FUNCTION_BLOCK "G274M_Code"
TITLE =G274M EXHAUST AIR LOUVER KILN 1
//COPYRIGHT:    (C) 2009  BUHLER AG, CH-9240 UZWIL, SWITZERLAND
//
//PRODUCT:      WinCoS_BIW01_09
//
//TITLE:        EXHAUST AIR LOUVER KILN 1
//                Machine group control
//                Maschinengruppensteuerung
//
//--------------------------------------------------------------------------------
//
//IDENT:        AUTHOR:             DEPT:                              DATE:
//
//P01_FB374.1.0 K.Renz              CSB41                              30.Sep.2009
//             1st Release
//
//--------------------------------------------------------------------------------
//
//PURPOSE:
//
//MANUAL :
//
//RESTRICTIONS:
//
//--------------------------------------------------------------------------------
AUTHOR : KR
FAMILY : USW
VERSION : 9.9


VAR
  Gr : "GCS7_GrpCtrlSub";	//Standard interface to group
  InOutValue1 : DINT ;	//Data for user
  InOutValue2 : DINT ;	//Data for user
  OutWayConflict : BOOL ;	//Data for user
  OutSelectionOk : BOOL ;	//Data for user
  CmdNewValue : BOOL ;	//Data for user
  CmdNewJob : BOOL ;	//Data for user
  OutCodeOK : BOOL ;	//Data for user
  InEndOfJob : BOOL ;	//Data for user
  staWayOk : BOOL ;	//Data for user
  EdgeStartRelease : BOOL ;	//Data for user
  USW8 : BOOL ;	//Data for user
  USW9 : BOOL ;	//Data for user
  USW10 : BOOL ;	//Data for user
  USW11 : BOOL ;	//Data for user
  USW12 : BOOL ;	//Data for user
  USW13 : BOOL ;	//Data for user
  USW14 : BOOL ;	//Data for user
  USW15 : BOOL ;	//Data for user
END_VAR
VAR_TEMP
  tmpEnable : BOOL ;
  tmpFlag : BOOL ;
  tmpCmdNext : BOOL ;
  tmpLocal : BOOL ;
  tmpAspOk : BOOL ;
  tmpHWStop : BOOL ;
  tmpInstanzDBNo : INT ;
END_VAR
BEGIN
NETWORK
TITLE =



NETWORK
TITLE =Read command from group control
//Parameter
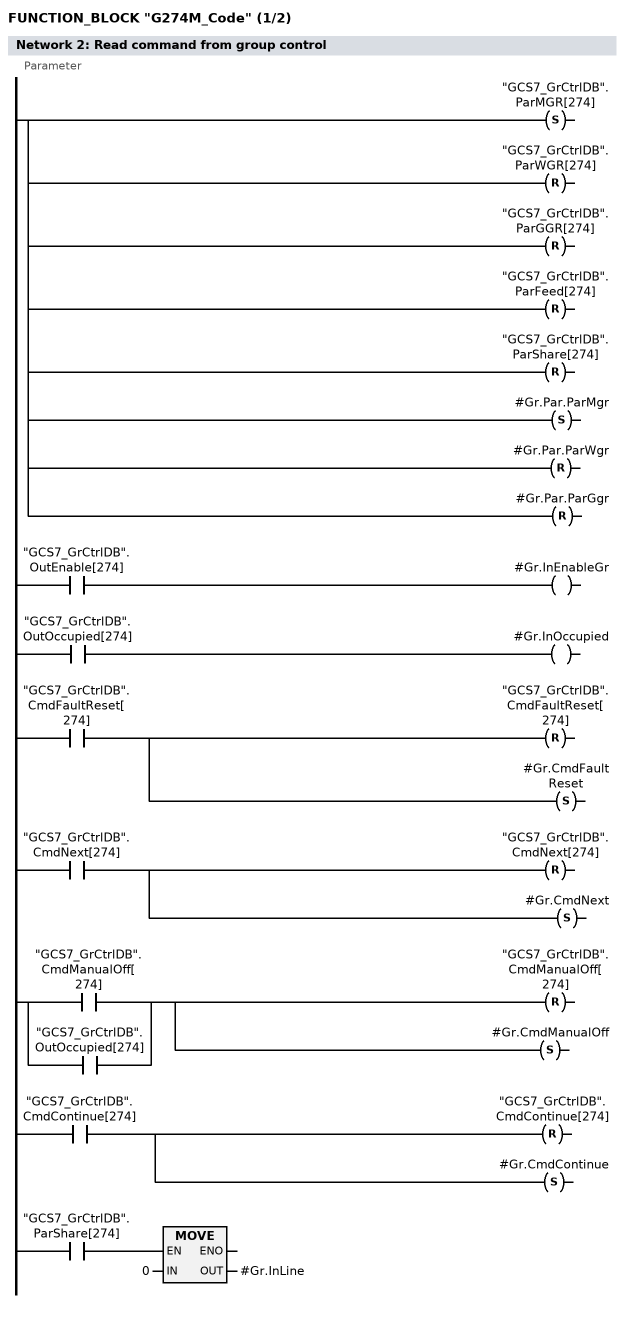
      SET   ;
      S     "GCS7_GrCtrlDB".ParMGR[274];
      R     "GCS7_GrCtrlDB".ParWGR[274];
      R     "GCS7_GrCtrlDB".ParGGR[274];
      R     "GCS7_GrCtrlDB".ParFeed[274];
      R     "GCS7_GrCtrlDB".ParShare[274];
      S     #Gr.Par.ParMgr;
      R     #Gr.Par.ParWgr;
      R     #Gr.Par.ParGgr;
//Command
      U     "GCS7_GrCtrlDB".OutEnable[274];
      =     #Gr.InEnableGr;
      U     "GCS7_GrCtrlDB".OutOccupied[274];
      =     #Gr.InOccupied;
      U     "GCS7_GrCtrlDB".CmdFaultReset[274];
      R     "GCS7_GrCtrlDB".CmdFaultReset[274];
      S     #Gr.CmdFaultReset;
      U     "GCS7_GrCtrlDB".CmdNext[274];
      R     "GCS7_GrCtrlDB".CmdNext[274];
      S     #Gr.CmdNext;
      U     "GCS7_GrCtrlDB".CmdManualOff[274];
      O     "GCS7_GrCtrlDB".OutOccupied[274];
      R     "GCS7_GrCtrlDB".CmdManualOff[274];
      S     #Gr.CmdManualOff;
      U     "GCS7_GrCtrlDB".CmdContinue[274];
      R     "GCS7_GrCtrlDB".CmdContinue[274];
      S     #Gr.CmdContinue;
//Init Line Number
      U     "GCS7_GrCtrlDB".ParShare[274];
      SPBN  WE00;
      L     0;
      T     #Gr.InLine;
WE00: NOP   0;
NETWORK
TITLE =Call Methode Control
// 1. Handle Interface PCControl
// 2. Prepare mode --> ModePassive,ModeActive,ModeIdling
// 3. Reset global flags of the group
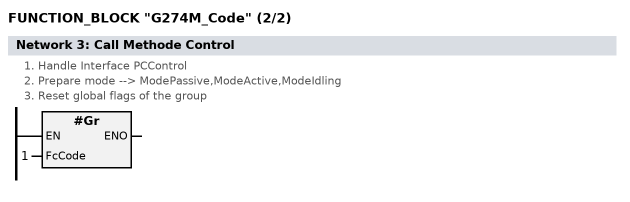
      CALL #Gr (
           FcCode                   := 1);
NETWORK
TITLE =Restart Idling Time

      L     #Gr.Par.ParIdling;
      L     2;
      >=I   ;
      SPB   IdTm;
      T     #Gr.Par.ParIdling;
IdTm: NOP   0;
      CLR   ;
      S     #Gr.CmdRestartIdling;
NETWORK
TITLE =Prepare global flags



NETWORK
TITLE =Set Pattern (Target position)



NETWORK
TITLE =Interlocking WayOk



NETWORK
TITLE =Interlocking Autostart

      CLR   ;
      R     #Gr.OutAutostart;
NETWORK
TITLE =Interlocking Enable
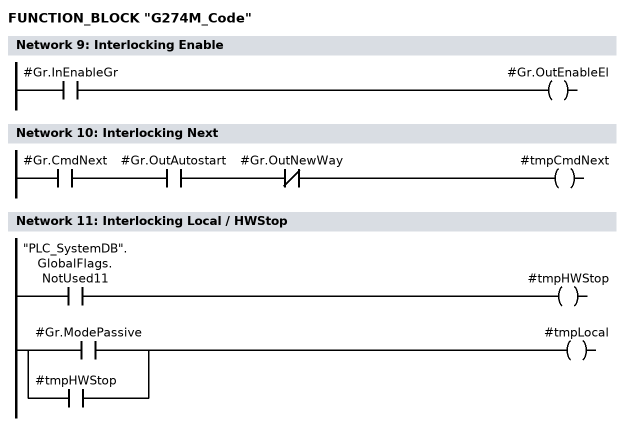

      U     #Gr.InEnableGr;
      =     #Gr.OutEnableEl;

NETWORK
TITLE =Interlocking Next

      U     #Gr.CmdNext;
      U     #Gr.OutAutostart;
      UN    #Gr.OutNewWay;
      =     #tmpCmdNext;

NETWORK
TITLE =Interlocking Local / HWStop

      U     "PLC_SystemDB".GlobalFlags.NotUsed11;
      =     #tmpHWStop;

      U     #Gr.ModePassive;
      O     #tmpHWStop;
      =     #tmpLocal;

NETWORK
TITLE =Test Fault

      CLR   ;
      =     #Gr.VarFault;
NETWORK
TITLE =Test Warning

      CLR   ;
      =     #Gr.OutWarning;
NETWORK
TITLE =Test Stopped

      UN    #Gr.VarFault;
      =     #Gr.VarStopped;
NETWORK
TITLE =Test Started

      CLR   ;
      UN    #Gr.VarStopped;
      UN    #Gr.VarFault;
      =     #Gr.VarStarted;
NETWORK
TITLE =Enable Previous Group
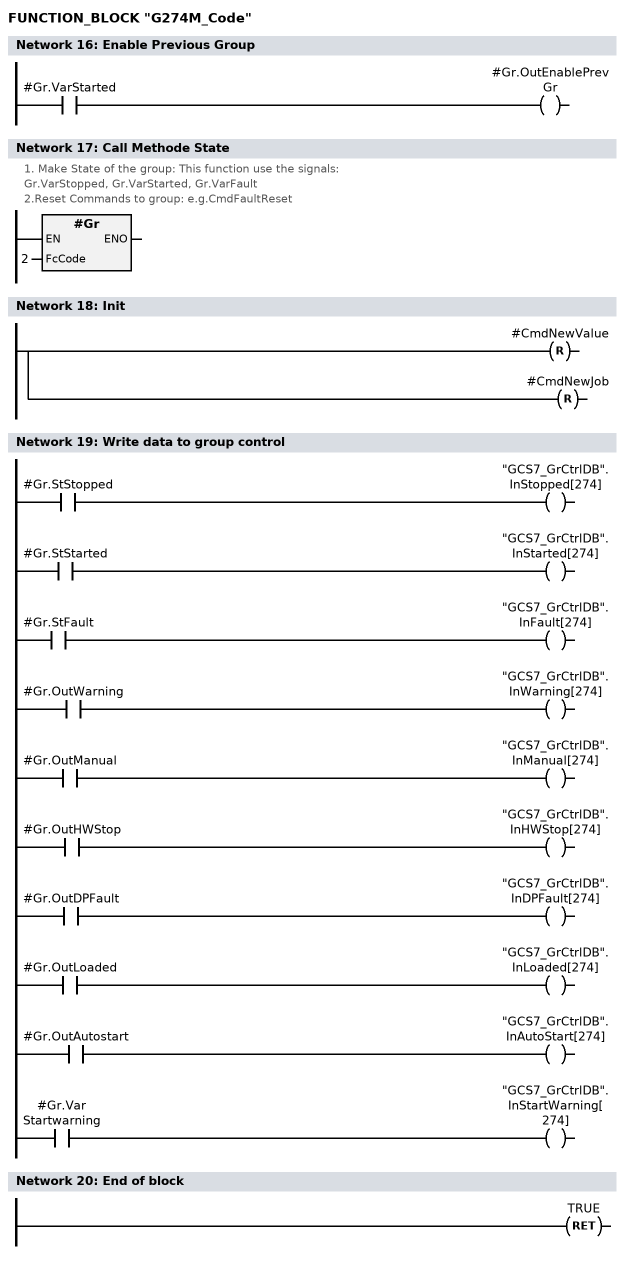

      U     #Gr.VarStarted;
      =     #Gr.OutEnablePrevGr;
NETWORK
TITLE =Call Methode State
//1. Make State of the group: This function use the signals:
//        Gr.VarStopped, Gr.VarStarted, Gr.VarFault
//2.Reset Commands to group: e.g.CmdFaultReset
      CALL #Gr (
           FcCode                   := 2);
NETWORK
TITLE =Init

      SET   ;
      R     #CmdNewValue;
      R     #CmdNewJob;
NETWORK
TITLE =Write data to group control

      U     #Gr.StStopped;
      =     "GCS7_GrCtrlDB".InStopped[274];
      U     #Gr.StStarted;
      =     "GCS7_GrCtrlDB".InStarted[274];
      U     #Gr.StFault;
      =     "GCS7_GrCtrlDB".InFault[274];
      U     #Gr.OutWarning;
      =     "GCS7_GrCtrlDB".InWarning[274];
      U     #Gr.OutManual;
      =     "GCS7_GrCtrlDB".InManual[274];
      U     #Gr.OutHWStop;
      =     "GCS7_GrCtrlDB".InHWStop[274];
      U     #Gr.OutDPFault;
      =     "GCS7_GrCtrlDB".InDPFault[274];
      U     #Gr.OutLoaded;
      =     "GCS7_GrCtrlDB".InLoaded[274];
      U     #Gr.OutAutostart;
      =     "GCS7_GrCtrlDB".InAutoStart[274];
      U     #Gr.VarStartwarning;
      =     "GCS7_GrCtrlDB".InStartWarning[274];
NETWORK
TITLE =End of block

      BE    ;

END_FUNCTION_BLOCK

